PROGRAM MAIN
VAR
	fbConveyor	:FB_Conveyor;
END_VAR

fbConveyor(stInput	:= GVL_IO.Conveyor_Inputs, stOutput=>GVL_IO.Conveyor_Outputs);

END_PROGRAM

(* stored: Version 1.1.0.1, ProductVersion 3.1.4024.16
   POU MAIN: Id {f6a867ed-f3fb-4c29-8585-1fbb6e585037}, SpecialFunc None *)
